(* IEC 61131-3 sources: AXOpen/src/inspectors/ctrl/src/AxoDigitalInspector, 3 files *)

(* ---- IAxoDigitalInspector.st ---- *)
USING AXOpen.Core;
NAMESPACE AXOpen.Inspectors
    INTERFACE IAxoDigitalInspector

        METHOD Inspect : IInspector
            VAR_INPUT
                _parent: IAxoObject;
                inData : REF_TO AxoDigitalInspectorData;
                Status : BOOL;
            END_VAR
        END_METHOD

    END_INTERFACE
END_NAMESPACE

(* ---- AxoDigitalInspector.st ---- *)
NAMESPACE AXOpen.Inspectors

    /// <summary>
    /// Class representing inspection of bool value.
    /// </summary>
    {S7.extern=ReadWrite}
    CLASS AxoDigitalInspector EXTENDS AxoInspector IMPLEMENTS IAxoDigitalInspector

        VAR PRIVATE
            _data : REF_TO AxoDigitalInspectorData;
        END_VAR

        /// <summary>
        /// Inspection method, which contains main logic of inspection.
        /// </summary>
        METHOD PUBLIC Inspect : IInspector
            VAR_INPUT
                _parent: AXOpen.Core.IAxoObject;
                inData : REF_TO AxoDigitalInspectorData;
                Status : BOOL;
            END_VAR

            _data := inData;

            THIS.Initialize(_parent);
            _inspectorTask.Initialize(_parent);

            //return this instance
            Inspect := THIS;

            // set task inspection data, pass a reference (an address)
            // REF(_data) will get a reference of _data variable (like & in C)
            _inspectorTask.SetInspectionData(_data);

            //here i should check, if data are overinspected
            IF(THIS.IsOverInspected()) THEN
                RETURN;
            END_IF;

            //invoke inspection task
            _inspectorTask.Invoke();

            //execute inspection task
            IF (_inspectorTask.Execute()) THEN

                // if data are bypassed, skip inspection
                IF (_data^.IsByPassed) THEN

                    _data^.Result    := eInspectorResult#Bypassed;

                    _data^.TimeStamp := THIS.GetContext().GetRtc().NowUTC();

                    _inspectorTask.DoneWhen(TRUE);
                    RETURN;
                END_IF;

                //set timers
                _data^.Result := eInspectorResult#Running;
                _inspectorTask._failTimer.OnDelay(THIS.GetContext(), TRUE, _data^.FailTime);
                _inspectorTask._passTimer.OnDelay(THIS.GetContext(), Status = _data^.RequiredStatus, _data^.PassTime);

                _data^.DetectedStatus := Status;

                // if any timer is satisfied, end inspection
                IF(_inspectorTask._failTimer.output OR _inspectorTask._passTimer.output) THEN
                    _inspectorTask.DoneWhen(TRUE);
                    IF (_data^.Result = eInspectorResult#Failed) THEN
                        _data^.DetectedStatus := NOT _data^.RequiredStatus;
                    END_IF;
                    THIS.OnDone();
                END_IF;
            END_IF;
        END_METHOD

        ///<summary>
        /// If inspection fails, set result to data
        ///</summary>
        METHOD OnDone
            ;
        END_METHOD

        ///<summary>
        /// Set coordinator to this instance
        ///</summary>
        METHOD PUBLIC WithCoordinator : IAxoDigitalInspector
            VAR_INPUT
                inCoordinator : AXOpen.Core.IAxoCoordinator;
            END_VAR

            _coordinator := inCoordinator;
            THIS._WithCoordinator(inCoordinator);

            WithCoordinator := THIS;
        END_METHOD

        ///<summary>
        /// Set coordinator to this instance
        ///</summary>
        METHOD PUBLIC Data : REF_TO AxoDigitalInspectorData

            Data := REF(_data^);
        END_METHOD

    END_CLASS
END_NAMESPACE

(* ---- AxoDigitalInspectorData.st ---- *)
NAMESPACE AXOpen.Inspectors

    ///<summary>
    /// Data subjected to each digital inspector instance.
    ///</summary>
    {S7.extern=ReadWrite}
    CLASS AxoDigitalInspectorData EXTENDS AxoInspectorData

        VAR PUBLIC
            //<AxoDigitalInspectorDataDeclaration>
            {#ix-set:AttributeName = "<#Required#>"}
            RequiredStatus : BOOL;

            {#ix-attr:[ReadOnly()]}
            {#ix-set:AttributeName = "<#Detected#>"}
            DetectedStatus : BOOL;
            //</AxoDigitalInspectorDataDeclaration>

        END_VAR

    END_CLASS

END_NAMESPACE
